// TIA Portal project "SmartTraySort" (V17)

(* hardware
DEVICE "S7-1200 station_1"  S7-1200 Station
   slot 0: "Rack_0"  S7-1200 Rack  Rack  V1.0
   slot 1: "TraySort"  CPU 1214C DC/DC/DC  6ES7 214-1AG40-0XB0  V4.5
*)

// ===== PLC "TraySort"  CPU 1214C DC/DC/DC =====

VAR_GLOBAL   // PLC tag table "Default tag table"
   "Axis_X_Pulse" AT %Q0.0 : Bool;
   "Axis_X_Direction" AT %Q0.1 : Bool;
   "Axis_Y_Pulse" AT %Q0.2 : Bool;
   "Axis_Y_Direction" AT %Q0.3 : Bool;
   "Axis_Z_Pulse" AT %Q0.6 : Bool;
   "Axis_Z_Direction" AT %Q0.7 : Bool;
   "Tag__639232821342344062" AT %I0.0 : Bool;
   "Axis_Z_Homing switch" AT %I0.1 : Bool;
END_VAR

TYPE "typSlot"
// ============================================================================
//   01_Types.scl  -  Khai bao kieu du lieu (UDT)
//   Project: SmartTraySort  |  S7-1200 CPU 1214C DC/DC/DC + TIA Portal V17
// 
//   BA TRUC:
//      Axis_X  ngang qua lai       driver HBS86H      (hybrid servo vong kin)
//      Axis_Y  lat trai phai +-60  driver ASD556R-LW  (buoc 2 pha)
//      Axis_Z  len xuong           driver 3DH583      (buoc 3 pha)
// 
//   Luoi 20 khay nam tren mat phang dung: X la cot trai/phai, Z la hang cao/thap.
//   Truc Y khong tham gia dinh vi khay, no chi lat khay ra hai ben.
// 
//   Kien truc: Orange Pi giu UI + luu do, PLC chi nhan lenh va thuc thi chuyen dong
//   Import: External source files -> Generate blocks from source
//   LUU Y: file .scl chi dung ky tu ASCII (khong dau) de TIA khong loi encoding
//  ============================================================================
//  Vi sao Real chu khong phai LReal:
//    1. Lenh Motion Control cua S7-1200 (MC_MoveAbsolute, MC_Home, MC_MoveJog)
//       nhan Real. Khai LReal thi den luc dung van phai cat bot - do chinh xac
//       thua bi vut di ngay tai cho, chi to them mot dong doi kieu.
//    2. Real cho ~7 chu so co nghia: o hanh trinh 1250 mm la phan giai duoi
//       0.001 mm, min hon buoc co khi (640 xung/mm ~ 0.0016 mm/xung) nhieu lan.
//    3. Quan trong nhat: mang 500 o x 12 byte = 6 000 byte, LOT vao 10 240 byte
//       bo nho luu khi mat dien cua S7-1200. Neu de LReal thi mot o ton 24 byte,
//       ca mang 12 000 byte - vuot tran, khong tick Retain duoc, va PLC se quen
//       sach bang toa do moi lan mat dien.
   STRUCT
      X : Real;   // vi tri ngang cua khay (mm)
      Z : Real;   // do cao cua khay (mm)
      Dir : Int;   // chieu lat cua khay nay: +1 = lat sang PHAI (+Y) -1 = lat sang TRAI (-Y) 0 = khong lat
   END_STRUCT;
END_TYPE

TYPE "typTray"
// ----------------------------------------------------------------------------
//  Bang du lieu may: 20 khay + tham so van hanh.
//  Tat ca deu chinh duoc luc dang chay, khong can sua chuong trinh.
//  ----------------------------------------------------------------------------
   STRUCT
      Pos : Array[1..500] of "typSlot";
      SlotCount : Int := 20;   // so ro dang dung, 1..500 --- VI TRI CHO = TRAM NAP --- Nam o DAU hanh trinh truc X, ngoai ria gian khay - cho nguoi dung dung quet ma va dat vat len khay. Cung la diem lay goc toa do, nen X = 0.
      HomeX : Real := 0.0;   // tram nap, dau truc X (mm)
      HomeY : Real := 0.0;   // goc giua cua truc lat (do)
      HomeZ : Real := 0.0;   // do cao cho cua truc len xuong (mm) --- toc do chay tu dong ---
      VelX : Real := 80.0;   // mm/s
      VelY : Real := 200.0;   // do/s - truc lat
      VelZ : Real := 60.0;   // mm/s - truc len xuong, cham hon vi chong trong luc --- toc do jog tay ---
      JogVelX : Real := 10.0;
      JogVelY : Real := 20.0;
      JogVelZ : Real := 10.0;
      JogMaxTime : Time := T#5S;   // AN TOAN: gioi han thoi gian jog lien tuc. Orange Pi giu bit jog roi rot mang thi truc tu dung sau khoang thoi gian nay.
      DwellTime : Time := T#1S;   // dung yen tai khay cho het rung truoc khi lat --- tham so buoc LAT (truc Y) ---
      TiltAngle : Real := 60.0;   // goc lat (do): sang phai = +60, sang trai = -60
      TiltHold : Time := T#1S;   // thoi gian giu o goc lat truoc khi tra ve
      TiltCount : Int := 1;   // so lan lat. Dat 0 = bo qua buoc lat
      TiltVel : Real := 200.0;   // toc do lat (do/s) --- 2 tham so de chuyen giua MO PHONG va MAY THAT ---
      HomeMode : Int := 0;   // 0 = set thang vi tri hien tai = 0 (dung cho PLCSIM, khong can cong tac Home) 3 = active homing, chay tim cong tac Home (may that)
      UseModbus : Bool := TRUE;   // TRUE = bat MB_SERVER, dung cho CPU that FALSE = tat di khi quay lai chay PLCSIM (PLCSIM khong mo duoc cong TCP that) --- duong di --- TRUE = chay ngang va len xuong CUNG LUC. Thoi gian di = cai lau hon trong hai truc, thay vi cong don. Duong di thanh duong cheo. FALSE = chay xong ngang roi moi len xuong (cach cu). Bat lai neu phat hien mam quet trung cai gi tren duong cheo. Truc LAT luon phai o giua truoc khi di chuyen - viec do khong doi.
      SyncMove : Bool := TRUE;
      UseStopBtn : Bool := FALSE;   // FALSE = bo qua nut DUNG cung o %I0.0 (mo phong / chua dau nut nao) TRUE = doc that %I0.0. Nut phai la tiep diem THUONG DONG: nha = co dien = cho chay, nhan hay dut day = dung. Bat TRUE ma chua dau day thi may nam im - dung, do la dung y.
   END_STRUCT;
END_TYPE

TYPE "typIF"
// ----------------------------------------------------------------------------
//  Vung giao tiep voi Orange Pi (Modbus TCP) va HMI phu.
//  Layout byte co dinh -> DB tao tu UDT nay PHAI bo "Optimized block access".
// 
//   === ORANGE PI GHI XUONG (ghi tron khoi HR0..HR9 bang 1 lenh FC16) ===
//    Byte  0..1   Command      HR0    ma lenh, xem bang duoi
//    Byte  2..3   SelPos       HR1    so khay 1..SlotCount (lenh 13: la so luong)
//    Byte  4..5   CtrlBits     HR2    bit0 X+ / bit1 X- / bit2 Y+ / bit3 Y-
//                                     bit4 Z+ / bit5 Z- / bit8 CapDienTruc
//    Byte  6..7   CmdSeq       HR3    so thu tu lenh, client tu tang moi lan gui lenh moi
//    Byte  8..11  TargetX      HR4-5  vi tri ngang tu do (lenh 8) / toa do khay (lenh 11)
//    Byte 12..15  TargetY      HR6-7  goc lat tu do (lenh 10) / chieu lat (lenh 11)
//    Byte 16..19  TargetZ      HR8-9  do cao tu do (lenh 8) / do cao khay (lenh 11)
// 
//   === PLC TRA VE (Orange Pi chi doc) ===
//    Byte 20..21  StatusBits   HR10   bit0 Ready bit1 Busy bit2 Done bit3 Homed bit4 Error
//    Byte 22..23  StepNo       HR11   buoc hien tai cua may trang thai
//    Byte 24..25  ErrorID      HR12   ma loi Motion Control
//    Byte 26..27  AckSeq       HR13   echo CmdSeq khi PLC DA NHAN lenh
//    Byte 28..29  DoneSeq      HR14   CmdSeq cua lenh DA CHAY XONG
//    Byte 30..31  Result       HR15   ket qua lenh, xem bang duoi
//    Byte 32..35  ActX         HR16-17 vi tri thuc ngang (mm)
//    Byte 36..39  ActY         HR18-19 goc lat thuc (do)
//    Byte 40..43  ActZ         HR20-21 do cao thuc (mm)
//    Byte 44..45  CurSlot      HR22   khay dang chay toi
//    Byte 46..47  (du phong)   HR23
// 
//   === BANG MA LENH (Command) ===
//     0 = khong co lenh (PLC tu xoa ve 0 sau khi nhan)
//     1 = CHAY TU DONG: toi khay SelPos -> dung -> LAT dung ben -> ve cho
//     2 = chay Home (lay goc toa do ca 3 truc)
//     3 = dung khan
//     4 = xoa loi
//     5 = Teach: luu vi tri hien tai vao khay SelPos
//     6 = chi DI toi khay SelPos roi dung tai do (khong lat, khong ve)
//     7 = chi LAT tai cho, theo chieu cua khay SelPos
//     8 = di toi vi tri tu do TargetX / TargetZ
//     9 = ve vi tri cho (di chuyen, khong phai chay lay goc)
//    10 = lat truc Y toi goc TargetY (dung de can chinh co cau lat)
//    11 = GHI toa do khay SelPos = (TargetX, TargetZ), chieu lat lay tu dau cua TargetY
//         -> de Orange Pi day ca bang toa do xuong sau khi cau hinh tren web
//    12 = GHI vi tri cho = (TargetX, TargetY, TargetZ)
//    13 = GHI so ro dang dung: SlotCount := SelPos
//    14 = GHI mot tham so chay may: SelPos = ma tham so, TargetX = gia tri
//         1 VelX   2 VelY   3 VelZ   4 TiltAngle   5 TiltVel
//         6 DwellTime(ms)   7 TiltHold(ms)   8 TiltCount
//         9 JogVelX  10 JogVelY  11 JogVelZ
//         -> vi tri cho khong o goc toa do ma o giua gian khay, noi lap cam bien
// 
//   === BANG KET QUA (Result) ===
//     0 = chua chay lenh nao
//     1 = dang chay
//     2 = hoan thanh tot
//     3 = bi dung giua chung (lenh Stop)
//     4 = loi
//     5 = lenh hoac tham so khong hop le / may chua san sang
//  ----------------------------------------------------------------------------
   STRUCT
      Command : Word;
      SelPos : Int;
      CtrlBits : Word;
      CmdSeq : Word;
      TargetX : Real;
      TargetY : Real;
      TargetZ : Real;   // --- PLC tra ve ---
      StatusBits : Word;
      StepNo : Int;
      ErrorID : Word;
      AckSeq : Word;
      DoneSeq : Word;
      Result : Word;
      ActX : Real;
      ActY : Real;
      ActZ : Real;
      CurSlot : Int;
      Spare1 : Int;
   END_STRUCT;
END_TYPE

DATA_BLOCK "DB_TrayTable"   // DB4
{ S7_Optimized_Access := 'TRUE' }
VERSION : 0.6
// ============================================================================
//   02_DB_TrayTable.scl  -  Bang toa do ro + tham so may
//   SINH TU CONG THUC, dung sua tay.
//   RETAIN: TICK HET, ca mang Pos.
//   Khoi nay khai bang KIEU ("typTray") nen ca DB la mot the hien cua UDT - TIA
//   chi dat Retain cho CA KHOI, khong tach duoc tung bien (bo tick mot o la bo
//   sach, khong phai loi).
//   Tick het van lot: toa do la Real nen mot o ton 12 byte,
//   500 o = 6 000 byte, con tran bo nho luu khi mat dien cua S7-1200 la 10 240
//   byte. (Neu de LReal thi mot o 24 byte, ca mang 12 000 byte - vuot tran,
//   download se bao "retentive memory exceeded". Do la ly do doi sang Real.)
// 
//   Nho Retain, BANG TOA DO LA CUA PLC: mat dien bat lai van con nguyen, khong
//   phu thuoc server co dang chay hay khong. Server chi day bang xuong khi nguoi
//   dung bam Luu cau hinh, va mot lan nua sau khi vua nap lai khoi trong TIA
//   (luc do DB tro ve gia tri khoi tao, Retain khong do duoc) - xem resync_plc
//   trong orangepi/app/main.py.
// 
//   So ro KHONG co dinh. No la ket qua tinh tu hanh trinh hai truc va kich
//   thuoc mot cai ro:
//      dem cot   : buoc chat nhat = ro dai 200 + khe toi thieu 10 = 210 mm
//                  hanh trinh X 1250 mm  ->  5 cot
//      dat toa do: trai deu ra cho mep ro cuoi cham dung 1250 mm,
//                  nen buoc that la 237.5 mm, khe ho that 37.5 mm
//      buoc hang : thanh ro 60 + nang khay 90 + khe ho 30 = 180 mm
//                  hanh trinh Z 400 mm  ->  2 hang (chua 20 mm le gioi han)
//      => 2 hang x 5 cot x 2 ben = 20 ro
// 
//   Ro to hon -> it ro lai. Truc X dai ra -> them ro. Web tinh lai roi day ca
//   bang lan SlotCount xuong day, khong phai sua file nay.
// 
//   Bo cuc: hai day ro nam hai ben duong ray, ban chay o giua. Cung mot vi tri X
//   phuc vu ca hai ben, chi khac chieu lat.
//   Danh so chay tu hang TREN xuong, moi hang het ben PHAI roi toi ben TRAI.
// 
//   Z KHONG phai do cao mieng ro. Ro dat sat hai ben ray nen khay phai dung CAO
//   HON mieng ro 90 mm thi vat moi roi lot vao trong chu khong dap vao thanh.
// 
//   Tram nap o X = 5, ngoai ria. Khong dat dung 0: 0 la gioi han phan mem,
//   do trung vach la PLC bao loi.
//  ============================================================================
BEGIN
   HomeX := 5.0;
   HomeZ := 5.0;
   Pos[1].X := 200.0;
   Pos[1].Z := 370.0;
   Pos[1].Dir := 1;
   Pos[2].X := 437.5;
   Pos[2].Z := 370.0;
   Pos[2].Dir := 1;
   Pos[3].X := 675.0;
   Pos[3].Z := 370.0;
   Pos[3].Dir := 1;
   Pos[4].X := 912.5;
   Pos[4].Z := 370.0;
   Pos[4].Dir := 1;
   Pos[5].X := 1150.0;
   Pos[5].Z := 370.0;
   Pos[5].Dir := 1;
   Pos[6].X := 200.0;
   Pos[6].Z := 370.0;
   Pos[6].Dir := -1;
   Pos[7].X := 437.5;
   Pos[7].Z := 370.0;
   Pos[7].Dir := -1;
   Pos[8].X := 675.0;
   Pos[8].Z := 370.0;
   Pos[8].Dir := -1;
   Pos[9].X := 912.5;
   Pos[9].Z := 370.0;
   Pos[9].Dir := -1;
   Pos[10].X := 1150.0;
   Pos[10].Z := 370.0;
   Pos[10].Dir := -1;
   Pos[11].X := 200.0;
   Pos[11].Z := 190.0;
   Pos[11].Dir := 1;
   Pos[12].X := 437.5;
   Pos[12].Z := 190.0;
   Pos[12].Dir := 1;
   Pos[13].X := 675.0;
   Pos[13].Z := 190.0;
   Pos[13].Dir := 1;
   Pos[14].X := 912.5;
   Pos[14].Z := 190.0;
   Pos[14].Dir := 1;
   Pos[15].X := 1150.0;
   Pos[15].Z := 190.0;
   Pos[15].Dir := 1;
   Pos[16].X := 200.0;
   Pos[16].Z := 190.0;
   Pos[16].Dir := -1;
   Pos[17].X := 437.5;
   Pos[17].Z := 190.0;
   Pos[17].Dir := -1;
   Pos[18].X := 675.0;
   Pos[18].Z := 190.0;
   Pos[18].Dir := -1;
   Pos[19].X := 912.5;
   Pos[19].Z := 190.0;
   Pos[19].Dir := -1;
   Pos[20].X := 1150.0;
   Pos[20].Z := 190.0;
   Pos[20].Dir := -1;
END_DATA_BLOCK

DATA_BLOCK "DB_Interface"   // DB5
{ S7_Optimized_Access := 'FALSE' }
VERSION : 0.1
// ============================================================================
//   03_DB_Interface.scl  -  Vung lenh / trang thai dung chung HMI + app ngoai
// 
//   QUAN TRONG: DB nay PHAI bo "Optimized block access"
//   (chuot phai vao DB -> Properties -> bo tick Optimized block access)
//   thi MB_SERVER moi anh xa duoc thanh holding register va app ngoai moi doc duoc.
//   Neu chi dung HMI thi de optimized cung chay binh thuong.
//  ============================================================================
BEGIN
END_DATA_BLOCK

DATA_BLOCK "DB_XY_Tray"   // DB6
{ S7_Optimized_Access := 'TRUE' }
VERSION : 0.2
// ============================================================================
//   08_FC_Main.scl  -  Instance DB + khoi goi tong
// 
//   Trong OB1 (Main) chi can keo tha 1 lenh goi duy nhat:
//         "FC_Main"(HwSafeOK := TRUE)          <- khi mo phong
//         "FC_Main"(HwSafeOK := "I_EstopOK")   <- khi ra may that
// 
//   Nut DUNG cung nam o %I0.0 va DA duoc doc san trong khoi nay - OB1 khong phai
//   sua gi. Cong tac cua no la CONG TAC CHUYEN MACH: bat/tat bang
//         "DB_TrayTable".UseStopBtn
//      FALSE (mac dinh) : bo qua %I0.0, may chay nhu cu. Dung khi mo phong hoac
//                         khi chua dau nut nao vao.
//      TRUE             : doc that. Nut phai la tiep diem THUONG DONG - nha nut
//                         thi %I0.0 = 1 (cho chay), nhan nut hoac dut day thi
//                         %I0.0 = 0 va may dung ngay.
//   Bat TRUE ma quen dau day thi may khong nhuc nhich - do la dung, khong phai loi.
// 
//   Khong sinh de len OB1 co san de tranh mat code cu cua ban.
// 
//   DIEU KIEN: 3 Technology Object phai duoc tao truoc va dat ten dung la
//              "Axis_X" (ngang), "Axis_Y" (lat trai phai), "Axis_Z" (len xuong).
//              Sai ten la bao loi khi bien dich.
//  ============================================================================
// stored: InstanceOfName FB_XY_Tray
"FB_XY_Tray"
BEGIN
END_DATA_BLOCK

DATA_BLOCK "DB_ModbusIF"   // DB7
{ S7_Optimized_Access := 'TRUE' }
VERSION : 0.2
// stored: InstanceOfName FB_ModbusIF
"FB_ModbusIF"
BEGIN
END_DATA_BLOCK

DATA_BLOCK "Axis_X"   // DB1, Motion_DB
{ S7_Optimized_Access := 'TRUE' }
AUTHOR : SIMATIC
FAMILY : BasicMC
NAME : TO_PosAx
VERSION : 8.0
// stored: InstanceOfName TO_PositioningAxis
"TO_PositioningAxis"
BEGIN
   // Axis.LengthUnitNormalized.Distance = 1013
   // Axis.DirectionOutputEnabledCU = TRUE
   // Axis.OnlinePtoModeCU = 16#0000_0002
   // Axis.SelectedChannel2EnumCU = %Q0.1
   // Axis.SelectedChannel1EnumCU = %Q0.0
   // Pulse.MinDeltaDeltaFrequencyCU = 0.004
   // Pulse.MaxDeltaDeltaFrequencyCU = 1.0E+10
   // Pulse.MinDeltaFrequencyCU = 0.005
   // Pulse.MaxDeltaFrequencyCU = 9.5E+9
   // Pulse.MinFrequencyCU = 1.0
   // Pulse.MaxFrequencyCU = 100000.0
   // Pulse.OutputSourceCU = 16#0000_0000
   // Axis.SelectPTO = 0
END_DATA_BLOCK

DATA_BLOCK "Axis_Y"   // DB2, Motion_DB
{ S7_Optimized_Access := 'TRUE' }
AUTHOR : SIMATIC
FAMILY : BasicMC
NAME : TO_PosAx
VERSION : 8.0
// stored: InstanceOfName TO_PositioningAxis
"TO_PositioningAxis"
BEGIN
   // Axis.DirectionOutputEnabledCU = TRUE
   // Axis.LengthUnit.LastDistance = -1
   // Axis.OnlinePtoModeCU = 16#0000_0002
   // Axis.SelectedChannel2EnumCU = %Q0.7
   // Axis.SelectedChannel1EnumCU = %Q0.6
   // Pulse.MinDeltaDeltaFrequencyCU = 0.004
   // Pulse.MaxDeltaDeltaFrequencyCU = 1.0E+10
   // Pulse.MinDeltaFrequencyCU = 0.005
   // Pulse.MaxDeltaFrequencyCU = 9.5E+9
   // Pulse.MinFrequencyCU = 1.0
   // Pulse.MaxFrequencyCU = 30000.0
   // Pulse.OutputSourceCU = 16#0000_0000
   // Axis.SelectPTO = 1
   // Axis.OnlinePtoIndexCU = 1
END_DATA_BLOCK

DATA_BLOCK "Axis_Z"   // DB3, Motion_DB
{ S7_Optimized_Access := 'TRUE' }
AUTHOR : SIMATIC
FAMILY : BasicMC
NAME : TO_PosAx
VERSION : 8.0
// stored: InstanceOfName TO_PositioningAxis
"TO_PositioningAxis"
BEGIN
   // Axis.HomingReferencePointSwitch_AddressCU = %I0.1
   // Axis.LengthUnitNormalized.Distance = 1013
   // Axis.OnlinePtoModeCU = 16#0000_0002
   // Axis.DirectionOutputEnabledCU = TRUE
   // Axis.SelectedChannel2EnumCU = %Q0.3
   // Axis.SelectedChannel1EnumCU = %Q0.2
   // Pulse.MinDeltaDeltaFrequencyCU = 0.004
   // Pulse.MaxDeltaDeltaFrequencyCU = 1.0E+10
   // Pulse.MinDeltaFrequencyCU = 0.005
   // Pulse.MaxDeltaFrequencyCU = 9.5E+9
   // Pulse.MinFrequencyCU = 1.0
   // Pulse.MaxFrequencyCU = 100000.0
   // Pulse.OutputSourceCU = 16#0000_0000
   // Axis.SelectPTO = 2
   // Axis.OnlinePtoIndexCU = 2
END_DATA_BLOCK

FUNCTION_BLOCK "FB_XY_Tray"   // FB1, SCL
{ S7_Optimized_Access := 'TRUE' }
VERSION : 0.5
// ============================================================================
//   04_FB_XY_Tray.scl  -  May trang thai dieu khien 3 truc, 20 khay
//      Axis_X  ngang qua lai  |  Axis_Y  lat trai phai  |  Axis_Z  len xuong
// 
//   PLC chi la co cau chap hanh. Orange Pi gui 1 ma lenh kem so khay,
//   PLC tu tra bang toa do, tu tinh duong di, chay xong bao ket qua.
// 
//   Chu trinh lenh 1:
//      chay X va Z CUNG LUC toi khay -> dung yen cho het rung
//      -> LAT dung ben cua khay, giu, tra ve giua
//      -> Y ve giua -> Z va X CUNG LUC ve cho -> bao xong
// 
//   Hai truc X va Z chay song song vi chung nam tren hai kenh xung roi nhau,
//   hoan toan doc lap. Thoi gian di bang cai LAU HON trong hai truc chu khong
//   phai cong don. Muon quay lai kieu chay lan luot thi dat DB_TrayTable.SyncMove
//   := FALSE. Rieng truc LAT phai ve giua truoc khi di chuyen - dieu do khong
//   bao gio duoc bo, mam dang nghieng ma chay ngang la dap vao thanh ro.
// 
//   Cac lenh Motion Control (MC_*) duoc goi TAP TRUNG O CUOI than khoi, sau CASE.
//   Vi vay bit .Done cua chung ve o vong quet ke tiep - logic chuyen buoc da tinh den.
//  ============================================================================
   VAR_INPUT
      Enable : Bool;   // cap dien cho truc (MC_Power)
      CmdCode : Int;   // ma lenh da duoc kiem tra hop le, 0 = khong co lenh
      CmdPulse : Bool;   // TRUE dung 1 vong quet khi co lenh moi
      CmdSeq : Word;   // so thu tu lenh do Orange Pi cap
      SelPos : Int;   // so khay 1..20
      TargetX : Real;   // vi tri ngang tu do / toa do khay khi ghi bang
      TargetY : Real;   // goc lat tu do / chieu lat khi ghi bang
      TargetZ : Real;   // do cao tu do / do cao khay khi ghi bang
      JogXp : Bool;   // jog tay - giu la chay
      JogXn : Bool;
      JogYp : Bool;
      JogYn : Bool;
      JogZp : Bool;
      JogZn : Bool;   // Nut DUNG tren tu dien, tiep diem THUONG DONG: TRUE = nut dang nha, cho chay FALSE = dang nhan, HOAC dut day De mac dinh TRUE de mo phong khong can dau gi van chay duoc.
      StopOK : Bool := TRUE;
   END_VAR
   VAR_OUTPUT
      Ready : Bool;   // san sang nhan lenh moi
      Busy : Bool;   // dang chay
      Done : Bool;   // vua hoan thanh 1 chu trinh
      Homed : Bool;   // ca 3 truc da co goc toa do
      Error : Bool;
      ErrorID : Word;
      StepNo : Int;   // buoc hien tai
      ActX : Real;   // vi tri thuc ngang (mm)
      ActY : Real;   // goc lat thuc (do)
      ActZ : Real;   // do cao thuc (mm)
      AckSeq : Word;   // echo CmdSeq khi da nhan lenh
      DoneSeq : Word;   // CmdSeq cua lenh da chay xong
      Result : Word;   // 0 chua chay / 1 dang chay / 2 xong / 3 bi dung / 4 loi / 5 lenh sai
      CurSlot : Int;   // khay dang chay toi (0 = toa do tu do)
   END_VAR
   VAR_IN_OUT
      AxisX : TO_PositioningAxis;   // ngang qua lai
      AxisY : TO_PositioningAxis;   // lat trai phai
      AxisZ : TO_PositioningAxis;   // len xuong
      Tbl : "typTray";   // truyen vao "DB_TrayTable" --- instance cac lenh Motion Control ---
   END_VAR
   VAR
      mcPowerX : MC_Power;
      mcPowerY : MC_Power;
      mcPowerZ : MC_Power;
      mcResetX : MC_Reset;
      mcResetY : MC_Reset;
      mcResetZ : MC_Reset;
      mcHomeX : MC_Home;
      mcHomeY : MC_Home;
      mcHomeZ : MC_Home;
      mcAbsX : MC_MoveAbsolute;
      mcAbsY : MC_MoveAbsolute;
      mcAbsZ : MC_MoveAbsolute;
      mcJogX : MC_MoveJog;
      mcJogY : MC_MoveJog;
      mcJogZ : MC_MoveJog;
      mcHaltX : MC_Halt;
      mcHaltY : MC_Halt;
      mcHaltZ : MC_Halt;   // --- dong ho ---
      tDwell : TON_TIME;   // dung yen tai khay truoc khi lat
      tTilt : TON_TIME;   // giu o goc lat
      tJog : TON_TIME;   // gioi han thoi gian jog lien tuc (an toan mang)
      tReset : TON_TIME;   // gioi han thoi gian cho MC_Reset --- bien noi bo ---
      exX : Bool;   // co lenh chay tuyet doi tung truc
      exY : Bool;
      exZ : Bool;
      exHome : Bool;
      exReset : Bool;   // dang chay MC_Reset tren ca 3 truc Ca bang toa do lan cac bien o day deu la Real - dung kieu ma lenh Motion Control cua S7-1200 nhan. Nho vay khong con mot dong doi kieu nao trong khoi nay ngoai may cho doc ActualPosition tu Technology Object (rieng no la LReal). StepNo va Error la TRANG THAI, khong phai ngo ra. May trang thai doc lai chung moi vong quet, ma doc thang ngo ra thi TIA canh bao "might not be initialized". Giu ban that o day, cuoi khoi chep ra ngoai.
      "step" : Int;   // buoc hien tai cua may trang thai
      err : Bool;   // co loi dang treo
      posX : Real;   // dich den dang gui cho MC_MoveAbsolute
      posY : Real;
      posZ : Real;
      velXnow : Real;   // toc do dang dung cho lan chay nay
      velYnow : Real;
      velZnow : Real;
      tgtX : Real;   // dich cua chu trinh
      tgtY : Real;
      tgtZ : Real;
      tiltOut : Real;   // goc lat dich
      tiltDir : Int;   // +1 phai / -1 trai / 0 khong lat
      tiltN : Int;   // so lan lat con lai
      doTilt : Bool;   // chu trinh nay co lat khong
      doReturn : Bool;   // chu trinh nay co ve cho khong
      curSeq : Word;   // CmdSeq cua chu trinh dang chay
      jogOK : Bool;
   END_VAR
   VAR_TEMP
      stopNow : Bool;
   END_VAR
BEGIN


   // =========================================================================
   // 1. CAP DIEN CHO TRUC - phai goi moi vong quet
   // =========================================================================
   #mcPowerX(Axis := #AxisX,
             Enable := #Enable,
             StopMode := 0);
   #mcPowerY(Axis := #AxisY,
             Enable := #Enable,
             StopMode := 0);
   #mcPowerZ(Axis := #AxisZ,
             Enable := #Enable,
             StopMode := 0);

   // =========================================================================
   // 2. DOC TRANG THAI TRUC
   // =========================================================================
   #ActX := LREAL_TO_REAL(#AxisX.ActualPosition);
   #ActY := LREAL_TO_REAL(#AxisY.ActualPosition);
   #ActZ := LREAL_TO_REAL(#AxisZ.ActualPosition);
   #Homed := #AxisX.StatusBits.HomingDone AND #AxisY.StatusBits.HomingDone
   AND #AxisZ.StatusBits.HomingDone;
   #Busy := (#step <> 0) AND (#step < 900);
   #Ready := #mcPowerX.Status AND #mcPowerY.Status AND #mcPowerZ.Status AND #Homed
   AND (#step = 0) AND NOT #err;

   // toc do mac dinh cho vong quet nay, buoc lat se ghi de ben duoi
   #velXnow := #Tbl.VelX;
   #velYnow := #Tbl.VelY;
   #velZnow := #Tbl.VelZ;

   #stopNow := FALSE;

   // =========================================================================
   // 3. NHAN LENH TU ORANGE PI / HMI
   // =========================================================================
   IF #CmdPulse THEN
       #AckSeq := #CmdSeq;   // bao cho client biet lenh da toi noi

       CASE #CmdCode OF

           1:  // ---- CHAY TU DONG: toi khay -> dung -> lat -> ve cho ----
               IF #Ready AND (#SelPos >= 1) AND (#SelPos <= #Tbl.SlotCount) THEN
                   #curSeq := #CmdSeq;
                   #Result := 1;
                   #Done := FALSE;
                   #CurSlot := #SelPos;
                   #tgtX := #Tbl.Pos[#SelPos].X;
                   #tgtZ := #Tbl.Pos[#SelPos].Z;
                   #tiltDir := #Tbl.Pos[#SelPos].Dir;
                   #doTilt := TRUE;
                   #doReturn := TRUE;
                   #step := 10;
               ELSE
                   #Result := 5;
                   #DoneSeq := #CmdSeq;
               END_IF;

           2:  // ---- chay Home lay goc toa do ca 3 truc ----
               IF (#step = 0) AND NOT #err
                   AND #mcPowerX.Status AND #mcPowerY.Status AND #mcPowerZ.Status THEN
                   #curSeq := #CmdSeq;
                   #Result := 1;
                   #Done := FALSE;
                   #step := 5;
               ELSE
                   #Result := 5;
                   #DoneSeq := #CmdSeq;
               END_IF;

           3:  // ---- dung khan ----
               #stopNow := TRUE;

           4:  // ---- xoa loi ----
               //     Khong xoa ngay tai day. MC_Reset can vai vong quet moi xoa xong
               //     loi o Technology Object, nen phai co trang thai cho han hoi.
               IF #err OR (#step >= 900) THEN
                   #curSeq := #CmdSeq;
                   #Result := 1;
                   #exReset := TRUE;
                   #step := 950;
               ELSE
                   #Result := 2;              // dang khong co loi, coi nhu xong
                   #DoneSeq := #CmdSeq;
               END_IF;

           5:  // ---- Teach: luu vi tri hien tai vao khay SelPos ----
               IF (#step = 0) AND (#SelPos >= 1) AND (#SelPos <= #Tbl.SlotCount) THEN
                   // ActualPosition cua Technology Object la LReal, bang toa do la
                   // Real - phai cat ro rang, khong TIA canh bao mat do chinh xac.
                   #Tbl.Pos[#SelPos].X := LREAL_TO_REAL(#AxisX.ActualPosition);
                   #Tbl.Pos[#SelPos].Z := LREAL_TO_REAL(#AxisZ.ActualPosition);
                   #Result := 2;
                   #DoneSeq := #CmdSeq;
               ELSE
                   #Result := 5;
                   #DoneSeq := #CmdSeq;
               END_IF;

           6:  // ---- chi DI toi khay, dung tai do ----
               IF #Ready AND (#SelPos >= 1) AND (#SelPos <= #Tbl.SlotCount) THEN
                   #curSeq := #CmdSeq;
                   #Result := 1;
                   #Done := FALSE;
                   #CurSlot := #SelPos;
                   #tgtX := #Tbl.Pos[#SelPos].X;
                   #tgtZ := #Tbl.Pos[#SelPos].Z;
                   #doTilt := FALSE;
                   #doReturn := FALSE;
                   #step := 10;
               ELSE
                   #Result := 5;
                   #DoneSeq := #CmdSeq;
               END_IF;

           7:  // ---- chi LAT tai cho, theo chieu cua khay SelPos ----
               IF #Ready AND (#SelPos >= 1) AND (#SelPos <= #Tbl.SlotCount) THEN
                   #curSeq := #CmdSeq;
                   #Result := 1;
                   #Done := FALSE;
                   #tiltDir := #Tbl.Pos[#SelPos].Dir;
                   #doTilt := TRUE;
                   #doReturn := FALSE;
                   #step := 100;
               ELSE
                   #Result := 5;
                   #DoneSeq := #CmdSeq;
               END_IF;

           8:  // ---- di toi vi tri tu do do Orange Pi tinh ----
               IF #Ready THEN
                   #curSeq := #CmdSeq;
                   #Result := 1;
                   #Done := FALSE;
                   #CurSlot := 0;
                   #tgtX := #TargetX;
                   #tgtZ := #TargetZ;
                   #doTilt := FALSE;
                   #doReturn := FALSE;
                   #step := 10;
               ELSE
                   #Result := 5;
                   #DoneSeq := #CmdSeq;
               END_IF;

           9:  // ---- ve vi tri cho (di chuyen, khong phai lay goc) ----
               IF #Ready THEN
                   #curSeq := #CmdSeq;
                   #Result := 1;
                   #Done := FALSE;
                   #doTilt := FALSE;
                   #doReturn := TRUE;
                   #step := 195;
               ELSE
                   #Result := 5;
                   #DoneSeq := #CmdSeq;
               END_IF;

           10: // ---- lat truc Y toi goc tu do (can chinh co cau) ----
               IF #Ready THEN
                   #curSeq := #CmdSeq;
                   #Result := 1;
                   #Done := FALSE;
                   #tgtY := #TargetY;
                   #step := 300;
               ELSE
                   #Result := 5;
                   #DoneSeq := #CmdSeq;
               END_IF;

           11: // ---- GHI toa do khay tu web (khong chay may) ----
               //     TargetX = vi tri ngang, TargetZ = do cao,
               //     dau cua TargetY quyet dinh chieu lat
               // Chan tren la kich thuoc mang chu khong phai SlotCount: luc dang day
               // bang xuong, SlotCount cu co the con nho hon bang moi.
               IF (#step = 0) AND (#SelPos >= 1) AND (#SelPos <= 500) THEN
                   #Tbl.Pos[#SelPos].X := #TargetX;
                   #Tbl.Pos[#SelPos].Z := #TargetZ;
                   IF #TargetY > 0.0 THEN
                       #Tbl.Pos[#SelPos].Dir := 1;
                   ELSIF #TargetY < 0.0 THEN
                       #Tbl.Pos[#SelPos].Dir := -1;
                   ELSE
                       #Tbl.Pos[#SelPos].Dir := 0;
                   END_IF;
                   #Result := 2;
                   #DoneSeq := #CmdSeq;
               ELSE
                   #Result := 5;
                   #DoneSeq := #CmdSeq;
               END_IF;

           14: // ---- GHI mot tham so chay may ----
               //     SelPos = ma tham so, TargetX = gia tri. Mot lenh lo het moi
               //     tham so vo huong, khoi phai them ma lenh moi cho tung cai.
               IF #step = 0 THEN
                   // Toc do PHAI duong. Go nham so 0 tren web thi MC_MoveAbsolute /
                   // MC_MoveJog bao loi ngay lan chay dau va may dung giua chung,
                   // nen chan ngay tu day. Ma 1 2 3 5 9 10 11 deu la toc do;
                   // 4 (goc lat) duoc am, 6 7 8 duoc bang 0.
                   // Dat truoc la 2, nhanh ELSE se ghi de thanh 5 neu ma tham so la.
                   // KHONG duoc doc lai #Result de suy ra ket qua: no la bien tinh,
                   // con giu gia tri cua lenh TRUOC do.
                   #Result := 2;
                   IF ((#SelPos <= 3) OR (#SelPos = 5) OR (#SelPos >= 9))
                       AND (#TargetX <= 0.0) THEN
                       #Result := 5;              // toc do 0 hay am -> tu choi
                   ELSE
                       CASE #SelPos OF
                           1:
                               #Tbl.VelX := #TargetX;        // mm/s
                           2:
                               #Tbl.VelY := #TargetX;        // do/s
                           3:
                               #Tbl.VelZ := #TargetX;        // mm/s
                           4:
                               #Tbl.TiltAngle := #TargetX;   // do
                           5:
                               #Tbl.TiltVel := #TargetX;     // do/s
                           6:
                               #Tbl.DwellTime := DINT_TO_TIME(REAL_TO_DINT(#TargetX));  // ms
                           7:
                               #Tbl.TiltHold := DINT_TO_TIME(REAL_TO_DINT(#TargetX));   // ms
                           8:
                               #Tbl.TiltCount := REAL_TO_INT(#TargetX);
                           9:
                               #Tbl.JogVelX := #TargetX;
                           10:
                               #Tbl.JogVelY := #TargetX;
                           11:
                               #Tbl.JogVelZ := #TargetX;
                           ELSE
                               #Result := 5;              // ma tham so la
                       END_CASE;
                   END_IF;
                   #DoneSeq := #CmdSeq;
               ELSE
                   #Result := 5;
                   #DoneSeq := #CmdSeq;
               END_IF;

           13: // ---- GHI so ro dang dung (SlotCount) tu web ----
               //     Bo cuc gian ro do server tinh ra tu hanh trinh va kich thuoc
               //     ro, nen so luong khong co dinh. SelPos mang so luong do.
               IF (#step = 0) AND (#SelPos >= 1) AND (#SelPos <= 500) THEN
                   #Tbl.SlotCount := #SelPos;
                   #Result := 2;
                   #DoneSeq := #CmdSeq;
               ELSE
                   #Result := 5;
                   #DoneSeq := #CmdSeq;
               END_IF;

           12: // ---- GHI vi tri cho (park) tu web ----
               //     Vi tri cho khong nhat thiet o goc toa do. May nay dat o giua gian
               //     khay, cho lap cam bien nhan biet vat.
               IF #step = 0 THEN
                   #Tbl.HomeX := #TargetX;
                   #Tbl.HomeY := #TargetY;
                   #Tbl.HomeZ := #TargetZ;
                   #Result := 2;
                   #DoneSeq := #CmdSeq;
               ELSE
                   #Result := 5;
                   #DoneSeq := #CmdSeq;
               END_IF;

           ELSE  // ma lenh khong ton tai
               #Result := 5;
               #DoneSeq := #CmdSeq;
       END_CASE;
   END_IF;

   // =========================================================================
   // 4. XOA LOI - chi goi lenh, viec ha co lam o buoc 950
   // =========================================================================
   #mcResetX(Axis := #AxisX,
             Execute := #exReset);
   #mcResetY(Axis := #AxisY,
             Execute := #exReset);
   #mcResetZ(Axis := #AxisZ,
             Execute := #exReset);
   #tReset(IN := #exReset,
           PT := T#5s);

   // =========================================================================
   // 5. DUNG KHAN - huy moi lenh dang chay
   // =========================================================================
   // Nut cung tren tu co quyen ngang lenh tu web. Bat theo MUC chu khong theo
   // suon: con giu nut thi con dung, nha ra moi chay tiep duoc.
   IF NOT #StopOK THEN
       #stopNow := TRUE;
   END_IF;

   IF #stopNow THEN
       IF #step <> 0 THEN
           #Result := 3;            // bao cho client biet chu trinh bi cat ngang
           #DoneSeq := #curSeq;
       END_IF;
       #exX := FALSE;
       #exY := FALSE;
       #exZ := FALSE;
       #exHome := FALSE;
       // Phai ha ca co Reset. Neu bam Dung dung luc dang o buoc 950 ma khong ha,
       // MC_Reset giu Execute = TRUE mai mai: lan xoa loi sau khong con suon len
       // nao de kich, may treo o buoc 950 va khong bao gio xoa duoc loi.
       #exReset := FALSE;
       #step := 0;
   END_IF;
   #mcHaltX(Axis := #AxisX,
            Execute := #stopNow);
   #mcHaltY(Axis := #AxisY,
            Execute := #stopNow);
   #mcHaltZ(Axis := #AxisZ,
            Execute := #stopNow);

   // =========================================================================
   // 6. JOG TAY - chi cho phep khi dang dung o buoc 0
   //    Co gioi han thoi gian: giu bit jog qua JogMaxTime thi tu cat.
   // =========================================================================
   #tJog(IN := (#JogXp OR #JogXn OR #JogYp OR #JogYn OR #JogZp OR #JogZn),
         PT := #Tbl.JogMaxTime);

   // Con giu nut Dung (hoac dut day) thi cam luon jog. Thieu dieu kien nay thi
   // buoc 5 ep #step := 0, ma jog chi doi #step = 0 - hoa ra bam Dung xong van
   // jog chay duoc, MC_MoveJog con doat quyen cua MC_Halt.
   #jogOK := (#step = 0) AND #mcPowerX.Status AND #mcPowerY.Status AND #mcPowerZ.Status
   AND NOT #err AND NOT #tJog.Q
   AND #StopOK AND NOT #stopNow;

   #mcJogX(Axis := #AxisX,
           JogForward := #JogXp AND #jogOK,
           JogBackward := #JogXn AND #jogOK,
           Velocity := #Tbl.JogVelX);
   #mcJogY(Axis := #AxisY,
           JogForward := #JogYp AND #jogOK,
           JogBackward := #JogYn AND #jogOK,
           Velocity := #Tbl.JogVelY);
   #mcJogZ(Axis := #AxisZ,
           JogForward := #JogZp AND #jogOK,
           JogBackward := #JogZn AND #jogOK,
           Velocity := #Tbl.JogVelZ);

   // =========================================================================
   // 7. MAY TRANG THAI
   // =========================================================================
   CASE #step OF

       0:  // ------- Cho lenh -------
           #exX := FALSE;
           #exY := FALSE;
           #exZ := FALSE;

       5:  // ------- Chay lay goc toa do ca 3 truc -------
           #exHome := TRUE;
           IF #mcHomeX.Done AND #mcHomeY.Done AND #mcHomeZ.Done THEN
               #exHome := FALSE;
               #Result := 2;
               #DoneSeq := #curSeq;
               #Done := TRUE;
               #step := 0;
           END_IF;

       10: // ------- Di toi khay: ngang + len xuong -------
           //  SyncMove = TRUE: kich ca hai truc trong cung mot vong quet roi cho
           //  ca hai bao xong. Hai truc nay chay tren hai kenh xung roi nhau nen
           //  hoan toan doc lap - thoi gian di bang cai LAU HON trong hai cai,
           //  chu khong phai cong don nhu truoc.
           //  Duong di la duong cheo, khong phai duong thang noi hai diem: moi
           //  truc chay theo toc do rieng cua no, xong truoc thi dung cho. S7-1200
           //  khong noi suy quy dao duoc, va o may nay cung khong can - can den
           //  dung toa do la du, di kieu gi khong quan trong.
           #posX := #tgtX;
           #posZ := #tgtZ;
           #exX := TRUE;
           #exZ := #Tbl.SyncMove;
           IF #Tbl.SyncMove THEN
               IF #mcAbsX.Done AND #mcAbsZ.Done THEN
                   #exX := FALSE;
                   #exZ := FALSE;
                   #step := 30;
               END_IF;
           ELSE
               IF #mcAbsX.Done THEN
                   #exX := FALSE;
                   #step := 20;
               END_IF;
           END_IF;

       20: // ------- Chay len xuong (chi dung khi SyncMove = FALSE) -------
           #posZ := #tgtZ;
           #exZ := TRUE;
           IF #mcAbsZ.Done THEN
               #exZ := FALSE;
               #step := 30;
           END_IF;

       30: // ------- Dung yen cho het rung (DwellTime) -------
           IF #tDwell.Q THEN
               IF #doTilt THEN
                   #step := 100;
               ELSIF #doReturn THEN
                   #step := 195;
               ELSE
                   #step := 220;
               END_IF;
           END_IF;

           // =====================================================================
           //  100..190  BUOC LAT - lat ve dung ben cua khay (Dir = +1 phai / -1 trai)
           // =====================================================================

       100: // ------- Chuan bi lat -------
           IF (#Tbl.TiltCount <= 0) OR (#tiltDir = 0) THEN
               #step := 190;                  // khong lat, bo qua
           ELSE
               #tiltN := #Tbl.TiltCount;
               #tiltOut := #Tbl.HomeY + INT_TO_REAL(#tiltDir) * #Tbl.TiltAngle;
               #step := 170;
           END_IF;

       170: // ------- Lat ra dung ben -------
           #posY := #tiltOut;
           #velYnow := #Tbl.TiltVel;
           #exY := TRUE;
           IF #mcAbsY.Done THEN
               #exY := FALSE;
               #step := 175;
           END_IF;

       175: // ------- Giu o goc lat (TiltHold) -------
           IF #tTilt.Q THEN
               #step := 180;
           END_IF;

       180: // ------- Tra truc lat ve giua -------
           #posY := #Tbl.HomeY;
           #velYnow := #Tbl.TiltVel;
           #exY := TRUE;
           IF #mcAbsY.Done THEN
               #exY := FALSE;
               #tiltN := #tiltN - 1;
               IF #tiltN > 0 THEN
                   #step := 170;               // lat tiep
               ELSE
                   #step := 190;
               END_IF;
           END_IF;

       190: // ------- Lat xong -------
           IF #doReturn THEN
               #step := 195;
           ELSE
               #step := 220;
           END_IF;

           // =====================================================================
           //  195..220  VE VI TRI CHO
           // =====================================================================

       195: // ------- Dua truc lat ve giua truoc khi di chuyen -------
           #posY := #Tbl.HomeY;
           #exY := TRUE;
           IF #mcAbsY.Done THEN
               #exY := FALSE;
               #step := 200;
           END_IF;

       200: // ------- Ve cho: len xuong + ngang -------
           //  Buoc 195 da dua truc lat ve giua roi, gio mam khong con thoi ra hai
           //  ben nua nen chay cheo an toan.
           #posZ := #Tbl.HomeZ;
           #posX := #Tbl.HomeX;
           #exZ := TRUE;
           #exX := #Tbl.SyncMove;
           IF #Tbl.SyncMove THEN
               IF #mcAbsZ.Done AND #mcAbsX.Done THEN
                   #exZ := FALSE;
                   #exX := FALSE;
                   #step := 220;
               END_IF;
           ELSE
               IF #mcAbsZ.Done THEN
                   #exZ := FALSE;
                   #step := 210;
               END_IF;
           END_IF;

       210: // ------- Chay ngang ve cho (chi dung khi SyncMove = FALSE) -------
           #posX := #Tbl.HomeX;
           #exX := TRUE;
           IF #mcAbsX.Done THEN
               #exX := FALSE;
               #step := 220;
           END_IF;

       220: // ------- Xong 1 chu trinh, bao ket qua cho Orange Pi -------
           #Done := TRUE;
           #Result := 2;
           #DoneSeq := #curSeq;
           #step := 0;

       300: // ------- Lat truc Y toi goc tu do (lenh 10) -------
           #posY := #tgtY;
           #exY := TRUE;
           IF #mcAbsY.Done THEN
               #exY := FALSE;
               #step := 220;
           END_IF;

       950: // ------- Dang xoa loi: cho MC_Reset xong o ca 3 truc -------
           IF #mcResetX.Done AND #mcResetY.Done AND #mcResetZ.Done THEN
               #exReset := FALSE;
               #err := FALSE;
               #ErrorID := W#16#0;
               #Result := 2;
               #DoneSeq := #curSeq;
               #step := 0;
           ELSIF #mcResetX.Error OR #mcResetY.Error OR #mcResetZ.Error OR #tReset.Q THEN
               #exReset := FALSE;          // xoa khong duoc, quay lai trang thai loi
               #Result := 4;
               #DoneSeq := #curSeq;
               #step := 900;
           END_IF;

       900: // ------- Loi: dung tai cho, cho lenh Reset -------
           #exX := FALSE;
           #exY := FALSE;
           #exZ := FALSE;
           #exHome := FALSE;

       ELSE  // buoc la -> ve 0 cho an toan
           #step := 0;
   END_CASE;

   // --- cac dong ho, goi sau CASE ---
   #tDwell(IN := (#step = 30),
           PT := #Tbl.DwellTime);
   #tTilt(IN := (#step = 175),
          PT := #Tbl.TiltHold);

   // =========================================================================
   // 8. BAT LOI TU CAC LENH MOTION CONTROL
   // =========================================================================
   // Trong luc dang chay MC_Reset (buoc 950) thi bo qua - neu khong, bit loi cu
   // chua kip tat se lap tuc dat lai StepNo := 900 va lenh xoa loi khong bao gio an.
   IF (#step <> 950)
       AND (#mcPowerX.Error OR #mcPowerY.Error OR #mcPowerZ.Error
       OR #mcHomeX.Error OR #mcHomeY.Error OR #mcHomeZ.Error
       OR #mcAbsX.Error OR #mcAbsY.Error OR #mcAbsZ.Error
       OR #mcJogX.Error OR #mcJogY.Error OR #mcJogZ.Error) THEN

       IF NOT #err THEN   // chi chot ma loi DAU TIEN, khong de loi sau de len
           #err := TRUE;
           IF #mcPowerX.Error THEN
               #ErrorID := #mcPowerX.ErrorID;
           ELSIF #mcPowerY.Error THEN
               #ErrorID := #mcPowerY.ErrorID;
           ELSIF #mcPowerZ.Error THEN
               #ErrorID := #mcPowerZ.ErrorID;
           ELSIF #mcHomeX.Error THEN
               #ErrorID := #mcHomeX.ErrorID;
           ELSIF #mcHomeY.Error THEN
               #ErrorID := #mcHomeY.ErrorID;
           ELSIF #mcHomeZ.Error THEN
               #ErrorID := #mcHomeZ.ErrorID;
           ELSIF #mcAbsX.Error THEN
               #ErrorID := #mcAbsX.ErrorID;
           ELSIF #mcAbsY.Error THEN
               #ErrorID := #mcAbsY.ErrorID;
           ELSIF #mcAbsZ.Error THEN
               #ErrorID := #mcAbsZ.ErrorID;
           ELSIF #mcJogX.Error THEN
               #ErrorID := #mcJogX.ErrorID;
           ELSIF #mcJogY.Error THEN
               #ErrorID := #mcJogY.ErrorID;
           ELSE
               #ErrorID := #mcJogZ.ErrorID;
           END_IF;

           IF #step <> 0 THEN     // dang chay do lenh nao thi bao truot lenh do
               #Result := 4;
               #DoneSeq := #curSeq;
           END_IF;
       END_IF;
       #step := 900;
   END_IF;

   // =========================================================================
   // 9. GOI CAC LENH DI CHUYEN (dat cuoi cung - xem ghi chu dau file)
   // =========================================================================
   // Position = toa do gan cho DIEM LAY GOC.
   //   HomeMode 0: diem lay goc chinh la cho may dang dung. May nay luon dung o
   //               VI TRI CHO khi lay goc, nen gan thang toa do vi tri cho vao day.
   //               Nho vay "lay goc" xong thi "ve cho cho" khong phai di dau ca.
   //   HomeMode 3: diem lay goc la cong tac Home. Khi lap cong tac roi thi doi
   //               HomeX/Y/Z thanh toa do that cua cong tac.
   #mcHomeX(Axis := #AxisX,
            Execute := #exHome,
            Position := #Tbl.HomeX,
            Mode := #Tbl.HomeMode);
   #mcHomeY(Axis := #AxisY,
            Execute := #exHome,
            Position := #Tbl.HomeY,
            Mode := #Tbl.HomeMode);
   #mcHomeZ(Axis := #AxisZ,
            Execute := #exHome,
            Position := #Tbl.HomeZ,
            Mode := #Tbl.HomeMode);

   #mcAbsX(Axis := #AxisX,
           Execute := #exX,
           Position := #posX,
           Velocity := #velXnow);
   #mcAbsY(Axis := #AxisY,
           Execute := #exY,
           Position := #posY,
           Velocity := #velYnow);
   #mcAbsZ(Axis := #AxisZ,
           Execute := #exZ,
           Position := #posZ,
           Velocity := #velZnow);

   // =========================================================================
   // 9. CHEP TRANG THAI RA NGO RA
   //    Lam o cuoi cung de gia tri gui ra luon la ket qua cua vong quet nay.
   // =========================================================================
   #StepNo := #step;
   #Error := #err;
END_FUNCTION_BLOCK

FUNCTION_BLOCK "FB_ModbusIF"   // FB2, SCL
{ S7_Optimized_Access := 'TRUE' }
VERSION : 0.1
// ============================================================================
//   07_FB_ModbusIF.scl  -  Modbus TCP Server cho app ngoai
// 
//   Anh xa ca "DB_Interface" thanh holding register HR0..HR23.
//   BAN DO DAY DU nam trong 01_Types.scl (phan mo ta "typIF") - do la ban duy
//   nhat dung, dung chep lai o day nua keo hai noi lech nhau:
//      HR0 Command | HR1 SelPos | HR2 CtrlBits | HR3 CmdSeq
//      HR4-5 TargetX | HR6-7 TargetY | HR8-9 TargetZ        <- client ghi
//      HR10 StatusBits | HR11 StepNo | HR12 ErrorID | HR13 AckSeq
//      HR14 DoneSeq | HR15 Result | HR16-17 ActX | HR18-19 ActY
//      HR20-21 ActZ | HR22 CurSlot | HR23 du phong          <- client doc
//   (Modbus Poll danh so tu 40001 -> HR0 = 40001)
// 
//   KHI CHAY PLCSIM: dat DB_TrayTable.UseModbus := FALSE.
//   PLCSIM khong mo duoc cong TCP that nen MB_SERVER se bao loi va lam nhieu
//   qua trinh test logic. Chi bat TRUE khi da download xuong CPU that.
// 
//   InterfaceId: la Hardware identifier cua cong PROFINET, thuong = 64.
//   Kiem tra dung gia tri o: Project tree -> PLC tags -> Show all tags
//   -> tab System constants -> tim "Local~PROFINET_interface_1".
//  ============================================================================
   VAR_INPUT
      Enable : Bool;   // noi toi DB_TrayTable.UseModbus
      InterfaceId : Hw_Any := 64;
      LocalPort : UInt := 502;
   END_VAR
   VAR_OUTPUT
      NDR : Bool;   // app vua ghi du lieu xuong
      DR : Bool;   // app vua doc du lieu len
      Error : Bool;
      Status : Word;
   END_VAR
   VAR_IN_OUT
      HoldReg : Variant;   // truyen vao "DB_Interface"
   END_VAR
   VAR
      srv : MB_SERVER;
      conn : TCON_IP_v4;
      initDone : Bool;
   END_VAR
BEGIN


   // --- nap tham so ket noi 1 lan duy nhat ---
   IF NOT #initDone THEN
       #conn.InterfaceId := #InterfaceId;
       #conn.ID := W#16#1;                  // so hieu ket noi, khong trung voi khoi khac
       #conn.ConnectionType := B#16#0B;     // 16#0B = 11 = TCP
       #conn.ActiveEstablished := FALSE;    // FALSE = PLC lam Server (thu dong cho)
       #conn.RemoteAddress.ADDR[1] := B#16#0;  // 0.0.0.0 = chap nhan moi client
       #conn.RemoteAddress.ADDR[2] := B#16#0;
       #conn.RemoteAddress.ADDR[3] := B#16#0;
       #conn.RemoteAddress.ADDR[4] := B#16#0;
       #conn.RemotePort := 0;
       #conn.LocalPort := #LocalPort;
       #initDone := TRUE;
   END_IF;

   // --- Modbus TCP server ---
   #srv(DISCONNECT := NOT #Enable,
        MB_HOLD_REG := #HoldReg,
        CONNECT := #conn,
        NDR => #NDR,
        DR => #DR,
        ERROR => #Error,
        STATUS => #Status);
END_FUNCTION_BLOCK

FUNCTION "FC_CmdDecode" : Void   // FC1, SCL
{ S7_Optimized_Access := 'TRUE' }
VERSION : 0.2
// ============================================================================
//   05_FC_CmdDecode.scl  -  Doc lenh tu Orange Pi / HMI
// 
//   Co che bat tay (quan trong khi master o xa qua mang LAN):
//     1. Orange Pi ghi 1 lan ca khoi HR0..HR7 (Command, SelPos, CtrlBits, CmdSeq,
//        TargetX, TargetY) bang lenh Modbus FC16 - ghi nhieu thanh ghi cung luc.
//     2. PLC thay Command <> 0 thi nhan lenh, chep CmdSeq sang AckSeq, roi
//        XOA Command ve 0. Client doc AckSeq = seq minh vua gui -> biet lenh da toi.
//     3. Chay xong PLC ghi DoneSeq = seq do va Result = ket qua.
//        Client doi DoneSeq = seq cua minh -> biet lenh da xong, khong can doan thoi gian.
// 
//   Nho vay lenh khong bao gio bi chay 2 lan, va client biet chinh xac trang thai
//   du mang co tre hay mat goi.
// 
//   Khong can bo bat suon (khong can bien Static) -> dung duoc FC.
//  ============================================================================
   VAR_OUTPUT
      CmdCode : Int;   // ma lenh 1..14, 0 = khong co lenh moi
      CmdPulse : Bool;   // TRUE dung 1 vong quet
      CmdSeq : Word;   // so thu tu lenh
      SelPos : Int;   // so o, da kiem tra; ngoai 1..500 tra ve 0
      TargetX : Real;
      TargetY : Real;
      TargetZ : Real;
      AxesEnable : Bool;   // bit8 CtrlBits - Orange Pi cho phep cap dien truc
      JogXp : Bool;
      JogXn : Bool;
      JogYp : Bool;
      JogYn : Bool;
      JogZp : Bool;
      JogZn : Bool;
   END_VAR
   VAR_IN_OUT
      IF_DB : "typIF";   // truyen vao "DB_Interface"
   END_VAR
BEGIN


   // --- co lenh moi hay khong ---
   IF #IF_DB.Command <> 0 THEN
       #CmdCode := WORD_TO_INT(#IF_DB.Command);
       #CmdPulse := TRUE;
       #IF_DB.Command := 0;         // ack: xoa ngay de chi tac dung 1 vong quet
   ELSE
       #CmdCode := 0;
       #CmdPulse := FALSE;
   END_IF;

   #CmdSeq := #IF_DB.CmdSeq;

   // --- kiem tra so o hop le ---
   // Chan tren la kich thuoc MANG (500), khong phai so ro dang dung. FB moi la
   // cho biet bang hien co bao nhieu ro that su, vi lenh 13 co the doi so do.
   IF (#IF_DB.SelPos >= 1) AND (#IF_DB.SelPos <= 500) THEN
       #SelPos := #IF_DB.SelPos;
   ELSE
       #SelPos := 0;                // 0 = khong hop le, FB se tra Result = 5
   END_IF;

   #TargetX := #IF_DB.TargetX;
   #TargetY := #IF_DB.TargetY;
   #TargetZ := #IF_DB.TargetZ;

   // --- cac bit tac dung lien tuc ---
   #JogXp := #IF_DB.CtrlBits.%X0;
   #JogXn := #IF_DB.CtrlBits.%X1;
   #JogYp := #IF_DB.CtrlBits.%X2;
   #JogYn := #IF_DB.CtrlBits.%X3;
   #JogZp := #IF_DB.CtrlBits.%X4;
   #JogZn := #IF_DB.CtrlBits.%X5;
   #AxesEnable := #IF_DB.CtrlBits.%X8;
END_FUNCTION

FUNCTION "FC_StatusPack" : Void   // FC2, SCL
{ S7_Optimized_Access := 'TRUE' }
VERSION : 0.2
// ============================================================================
//   06_FC_StatusPack.scl  -  Dong goi trang thai gui ve Orange Pi / HMI
//   Goi SAU FB_XY_Tray trong FC_Main de so lieu la cua vong quet hien tai.
//  ============================================================================
   VAR_INPUT
      Ready : Bool;
      Busy : Bool;
      Done : Bool;
      Homed : Bool;
      Error : Bool;
      ErrorID : Word;
      StepNo : Int;
      ActX : Real;
      ActY : Real;
      ActZ : Real;
      AckSeq : Word;
      DoneSeq : Word;
      Result : Word;
      CurSlot : Int;
   END_VAR
   VAR_IN_OUT
      IF_DB : "typIF";   // truyen vao "DB_Interface"
   END_VAR
BEGIN

   #IF_DB.StatusBits.%X0 := #Ready;
   #IF_DB.StatusBits.%X1 := #Busy;
   #IF_DB.StatusBits.%X2 := #Done;
   #IF_DB.StatusBits.%X3 := #Homed;
   #IF_DB.StatusBits.%X4 := #Error;

   #IF_DB.StepNo := #StepNo;
   #IF_DB.ErrorID := #ErrorID;
   #IF_DB.AckSeq := #AckSeq;
   #IF_DB.DoneSeq := #DoneSeq;
   #IF_DB.Result := #Result;
   #IF_DB.ActX := #ActX;
   #IF_DB.ActY := #ActY;
   #IF_DB.ActZ := #ActZ;
   #IF_DB.CurSlot := #CurSlot;
END_FUNCTION

FUNCTION "FC_Main" : Void   // FC3, SCL
{ S7_Optimized_Access := 'TRUE' }
VERSION : 0.3
   VAR_INPUT
      HwSafeOK : Bool;   // dieu kien an toan phan cung. Mo phong: dat TRUE. May that: noi vao tiep diem E-Stop OK / relay an toan.
   END_VAR
   VAR_TEMP
      cmdCode : Int;
      cmdPulse : Bool;
      cmdSeq : Word;
      selPos : Int;
      targetX : Real;
      targetY : Real;
      targetZ : Real;
      axesEn : Bool;
      jogXp : Bool;
      jogXn : Bool;
      jogYp : Bool;
      jogYn : Bool;
      jogZp : Bool;
      jogZn : Bool;
      enableAxes : Bool;
      stopOK : Bool;
   END_VAR
BEGIN


   // =========================================================================
   // 1. Doc lenh tu Orange Pi / HMI
   // =========================================================================
   "FC_CmdDecode"(CmdCode => #cmdCode,
                  CmdPulse => #cmdPulse,
                  CmdSeq => #cmdSeq,
                  SelPos => #selPos,
                  TargetX => #targetX,
                  TargetY => #targetY,
                  TargetZ => #targetZ,
                  AxesEnable => #axesEn,
                  JogXp => #jogXp,
                  JogXn => #jogXn,
                  JogYp => #jogYp,
                  JogYn => #jogYn,
                  JogZp => #jogZp,
                  JogZn => #jogZn,
                  IF_DB := "DB_Interface");

   // =========================================================================
   // 2. Dieu kien cap dien cho truc
   //    - Luon phai co dieu kien an toan phan cung.
   //    - Khi chay THAT (UseModbus = TRUE): Orange Pi phai chu dong bat bit8
   //      cua CtrlBits (gia tri 256) thi truc moi co dien. Master mat ket noi
   //      hay chua san sang thi truc khong tu nhien chay duoc.
   //    - Khi MO PHONG (UseModbus = FALSE): bo qua dieu kien tren cho de test.
   // =========================================================================
   #enableAxes := #HwSafeOK AND (#axesEn OR NOT "DB_TrayTable".UseModbus);

   // =========================================================================
   // 3. May trang thai dieu khien truc
   // =========================================================================
   // Nut DUNG cung doc thang tai day, khong bat OB1 phai sua.
   //   UseStopBtn = FALSE -> ve phai luon TRUE -> StopOK = TRUE -> chay binh thuong.
   //   UseStopBtn = TRUE  -> StopOK bam theo %I0.0 (tiep diem thuong dong).
   #stopOK := "Tag__639232821342344062" OR NOT "DB_TrayTable".UseStopBtn;

   "DB_XY_Tray"(Enable := #enableAxes,
                StopOK := #stopOK,
                CmdCode := #cmdCode,
                CmdPulse := #cmdPulse,
                CmdSeq := #cmdSeq,
                SelPos := #selPos,
                TargetX := #targetX,
                TargetY := #targetY,
                TargetZ := #targetZ,
                JogXp := #jogXp,
                JogXn := #jogXn,
                JogYp := #jogYp,
                JogYn := #jogYn,
                JogZp := #jogZp,
                JogZn := #jogZn,
                AxisX := "Axis_X",
                AxisY := "Axis_Y",
                AxisZ := "Axis_Z",
                Tbl := "DB_TrayTable");

   // =========================================================================
   // 4. Tra trang thai ve Orange Pi / HMI
   // =========================================================================
   "FC_StatusPack"(Ready := "DB_XY_Tray".Ready,
                   Busy := "DB_XY_Tray".Busy,
                   Done := "DB_XY_Tray".Done,
                   Homed := "DB_XY_Tray".Homed,
                   Error := "DB_XY_Tray".Error,
                   ErrorID := "DB_XY_Tray".ErrorID,
                   StepNo := "DB_XY_Tray".StepNo,
                   ActX := "DB_XY_Tray".ActX,
                   ActY := "DB_XY_Tray".ActY,
                   ActZ := "DB_XY_Tray".ActZ,
                   AckSeq := "DB_XY_Tray".AckSeq,
                   DoneSeq := "DB_XY_Tray".DoneSeq,
                   Result := "DB_XY_Tray".Result,
                   CurSlot := "DB_XY_Tray".CurSlot,
                   IF_DB := "DB_Interface");

   // =========================================================================
   // 5. Modbus TCP server cho Orange Pi
   //    Tu dong tat khi DB_TrayTable.UseModbus = FALSE (che do mo phong)
   // =========================================================================
   "DB_ModbusIF"(Enable := "DB_TrayTable".UseModbus,
                 InterfaceId := 64,
                 LocalPort := 502,
                 HoldReg := "DB_Interface");
END_FUNCTION

ORGANIZATION_BLOCK "Main"   // OB1, LAD, ProgramCycle
TITLE = "Main Program Sweep (Cycle)"
{ S7_Optimized_Access := 'TRUE' }
VERSION : 0.1
   VAR_INPUT
      Initial_Call : Bool;   // Initial call of this OB
      Remanence : Bool;   // =True, if remanent data are available
   END_VAR
BEGIN

REGION Network 1
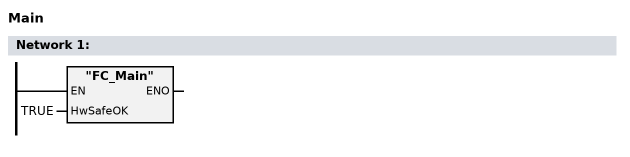
   RUNG wire#powerrail
      "FC_Main"(HwSafeOK := TRUE)
   END_RUNG
   // the same network as SCL:
   "FC_Main"(HwSafeOK := TRUE);
END_REGION
END_ORGANIZATION_BLOCK